SUBAPPLICATION SubApp_Retroreflective_Sensor (* Subapplication Type *)
  (* Standard: 61499-2 *)
  (* Version 1.0, 2022-10-10, AK123957 *)
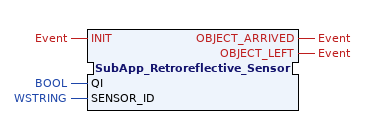
  EVENT_INPUT
    INIT;
  END_EVENT
  EVENT_OUTPUT
    OBJECT_ARRIVED;
    OBJECT_LEFT;
  END_EVENT
  VAR_INPUT
    QI : BOOL;
    SENSOR_ID : WSTRING;
  END_VAR
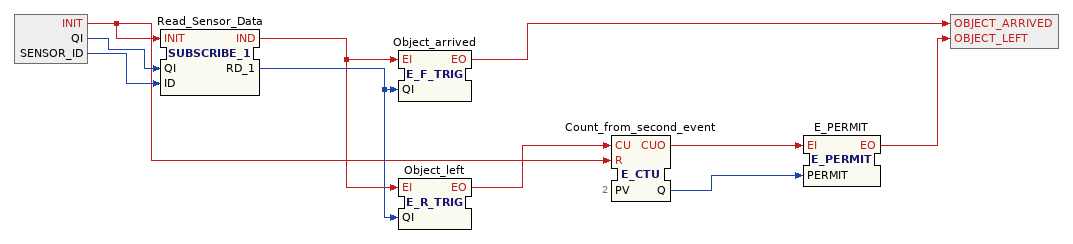
  FBS
    Object_left : E_R_TRIG;
    Read_Sensor_Data : SUBSCRIBE_1;
    Object_arrived : E_F_TRIG;
    Count_from_second_event : E_CTU(PV := 2);
    E_PERMIT : E_PERMIT;
  END_FBS
  EVENT_CONNECTIONS
    Read_Sensor_Data.IND TO Object_left.EI;
    Read_Sensor_Data.IND TO Object_arrived.EI;
    INIT TO Read_Sensor_Data.INIT;
    Object_arrived.EO TO OBJECT_ARRIVED;
    Count_from_second_event.CUO TO E_PERMIT.EI;
    Object_left.EO TO Count_from_second_event.CU;
    E_PERMIT.EO TO OBJECT_LEFT;
    INIT TO Count_from_second_event.R;
  END_CONNECTIONS
  DATA_CONNECTIONS
    Read_Sensor_Data.RD_1 TO Object_left.QI;
    Read_Sensor_Data.RD_1 TO Object_arrived.QI;
    QI TO Read_Sensor_Data.QI;
    SENSOR_ID TO Read_Sensor_Data.ID;
    Count_from_second_event.Q TO E_PERMIT.PERMIT;
  END_CONNECTIONS
END_SUBAPPLICATION
